// TIA Portal V20 export
FUNCTION_BLOCK "FB_GestionWorkingModes"   // FB94, SCL
{ S7_Optimized_Access := 'TRUE' }
// stored: MemoryReserve 100, SetENOAutomatically false
   VAR
      sMCP_KxxKeysDisable : Bool;
   END_VAR
BEGIN
   REGION Description header 
       //==================================================================================
       // POSALUX Swiss SA / (C) Copyright 2025
       //----------------------------------------------------------------------------------
       // Title: FB_GestionWorkingModes
       // Comment/Function: 
       // Author: Fabien WALDT
       // Engineering: TIA Portal v17
       //----------------------------------------------------------------------------------
       // Change log table:
       // Version  | Date     | Expert in charge | Changes applied
       // ---------|----------|------------------|-----------------------------------------
       // 00.00.01 | 20251218 | WFA              | First released version
       // =================================================================================
   END_REGION

   REGION Working Modes
       // MCP Keys Auto - Semi Auto disable
       "DB_McpKeyboardSignals".sK10_LoaderAuto.sKeyDisable := NOT "DB_WorkingModes".iChangeModeEnable OR #sMCP_KxxKeysDisable;
       "DB_McpKeyboardSignals".sK11_LoaderSemiAuto.sKeyDisable := NOT "DB_WorkingModes".iChangeModeEnable OR #sMCP_KxxKeysDisable;

       // Auto Mode Request
       IF "DB_McpKeyboardSignals".sK10_LoaderAuto.sKeySWTogglePositiveFront
           OR "DB_OPC_State".sRT_AutoReq.Q THEN
           "DB_WorkingModes".ioAutoReq := TRUE;
           "DB_McpKeyboardSignals".sK10_LoaderAuto.sKeySWToggleStatus := TRUE;
           "DB_McpKeyboardSignals".sK11_LoaderSemiAuto.sKeySWToggleStatus := FALSE;
       END_IF;

       // Semi Auto Mode Request
       IF "DB_McpKeyboardSignals".sK11_LoaderSemiAuto.sKeySWTogglePositiveFront
           OR "DB_OPC_State".sRT_SemiAutoReq.Q THEN
           "DB_WorkingModes".ioSemiAutoReq := TRUE;
           "DB_McpKeyboardSignals".sK10_LoaderAuto.sKeySWToggleStatus := FALSE;
           "DB_McpKeyboardSignals".sK11_LoaderSemiAuto.sKeySWToggleStatus := TRUE;
       END_IF;

       // Manu Mode Request
       IF ("DB_McpKeyboardSignals".sK11_LoaderSemiAuto.sKeySWToggleNegativeFront AND NOT "DB_McpKeyboardSignals".sK10_LoaderAuto.sKeySWToggleStatus)
           OR ("DB_McpKeyboardSignals".sK10_LoaderAuto.sKeySWToggleNegativeFront AND NOT "DB_McpKeyboardSignals".sK11_LoaderSemiAuto.sKeySWToggleStatus)
           OR "DB_OPC_State".sRT_ManuReq.Q THEN
           "DB_WorkingModes".ioManuReq := TRUE;
           "DB_McpKeyboardSignals".sK10_LoaderAuto.sKeySWToggleStatus := FALSE;
           "DB_McpKeyboardSignals".sK11_LoaderSemiAuto.sKeySWToggleStatus := FALSE;
       END_IF;

       "DB_WorkingModes"(ioEmptyingReq := "DB_HMISetting".WorkingMode.EmptyingReq,
                         ioAutoReq := "DB_WorkingModes".ioAutoReq,
                         ioSemiAutoReq := "DB_WorkingModes".ioSemiAutoReq,
                         ioManuReq := "DB_WorkingModes".ioManuReq,
                         iChangeModeEnable := NOT "DB_LoaderShuttle1".sMain.sInterface.SequenceRun
                         AND NOT "DB_LoaderShuttle2".sMain.sInterface.SequenceRun);

       IF "DB_PartManagement".sPosition.sMachineEmpty THEN
           "DB_HMISetting".WorkingMode.EmptyingReq := FALSE;
       END_IF;

       // Reset flags OPC
       "DB_OPC_State".sAutoReq := FALSE;
       "DB_OPC_State".sSemiAutoReq := FALSE;
       "DB_OPC_State".sManuReq := FALSE;
   END_REGION

   REGION Kxx Keys Disable
       IF #sMCP_KxxKeysDisable THEN
           "DB_McpKeyboardSignals".sK1_Powermeter.sKeyDisable := TRUE;
           "DB_McpKeyboardSignals".sK2_GasAssist.sKeyDisable := TRUE;
           "DB_McpKeyboardSignals".sK3_KeySaveParam.sKeyDisable := TRUE;
           "DB_McpKeyboardSignals".sK4_GripperUndrilledPart.sKeyDisable := TRUE;
           "DB_McpKeyboardSignals".sK5_GripperDrilledPart.sKeyDisable := TRUE;
           "DB_McpKeyboardSignals".sK6_SITestStop.sKeyDisable := TRUE;
           "DB_McpKeyboardSignals".sK7_FixtureClamp.sKeyDisable := TRUE;
           "DB_McpKeyboardSignals".sK8_FixtureVacuum.sKeyDisable := TRUE;
           "DB_McpKeyboardSignals".sK9_Aspiration.sKeyDisable := TRUE;
           "DB_McpKeyboardSignals".sK10_LoaderAuto.sKeyDisable := TRUE;
           "DB_McpKeyboardSignals".sK11_LoaderSemiAuto.sKeyDisable := TRUE;
           "DB_McpKeyboardSignals".sK12_ObservationCamera.sKeyDisable := TRUE;
           "DB_McpKeyboardSignals".sK13_MainDoor.sKeyDisable := TRUE;
           "DB_McpKeyboardSignals".sK14_WarmUp.sKeyDisable := TRUE;
           "DB_McpKeyboardSignals".sK15_MachineLight.sKeyDisable := TRUE;
       END_IF;
   END_REGION
END_FUNCTION_BLOCK
